REGION Network 2: Block description — Section 3 to 3.2
   // ▄▄▄▄▄▄▄▄▄▄▄▄▄▄▄▄▄▄▄▄▄▄▄▄▄▄▄▄▄▄▄▄▄▄▄▄▄▄▄▄▄▄▄▄
   // 3.     DETAILED BLOCK DESCRIPTION
   // 
   // 
   // This module, FC11001_StdDevValveIsol uses user data types to provide the primary interface to 
   // the module, it also uses direct digital signals to provide an interface for the position feedback 
   // signals and for the fault, safety and interlock signals. It also has a single output signal used to 
   // operate the valve. 
   // 
   // These are the formal module parameters: 
   // 
   //  ――――――――――――――――――――――――――――――――――――――――――
   //  PARAM         FUNCTION                    TYPE      IN-OUT 
   //  ――――――――――――――――――――――――――――――――――――――――――
   //  SYS_SIGNALS      Common system signals              UT21000    In
   //           logic and timing signals for parametric access
   // 
   //  FBK_OPEN     Optional open state positive feedback        Bool      In
   //           (1 = open, 0 = not open) If not required, set 
   //           permanently to _False
   // 
   //  FBK_CLOSED    Optional closed state positive feedback        Bool      In
   //           (1 = closed 0 = not closed) If not required, set 
   //           permanently to _False
   // 
   //  EXT_FAULT     Optional external fault signal for the device     Bool      In
   //           (1 = fault, 0 = healthy). If not required, set 
   //           permanently to _False
   // 
   //  E_STOP        Optional emergency stop (safety) signal        Bool      In
   //           (1 = emergency stop active, 0 = healthy) If not 
   //           required, set permanently to _False
   // 
   //  TRIP        Optional trip signal                  Bool      In
   //           (1 = trip condition active, 0 = healthy) If not 
   //           required, set permanently to _False
   // 
   //  INTERLOCK     Optional interlock signal               Bool      In
   //           (1 = interlock condition active, 0 = healthy) If 
   //           not required, set permanently to _False
   // 
   //  PERMISSIVE      Optional permissive signal             Bool      In
   //           (1 = permissive condition active, 0 = healthy) 
   //           If not required, set permanently to _False
   // 
   //  STATIC_DATA     Data structure that holds the configuration data     UT11001    In
   //           for the device (normally open/closed, limit switch 
   //           and interlock configuration &c.)
   // 
   //  DYNAMIC_DATA      Data structure that holds the live data for the       UT31001    InOut
   //           device (its mode, status and messages and 
   //           any other dynamic information required by the 
   //           module)
   // 
   //  OPERATE        Output to drive the valve to a particular state    Bool      Out
   //           (1 = energised state, 0 = deenergised state)
   //  ――――――――――――――――――――――――――――――――――――――――――
   // 
   // FBK_OPEN, FBK_CLOSED and EXT_FAULT parameters are input signals provided directly from the 
   // device itself (via digital input cards). The OPERATE signal is an output signal (via a digital output 
   // card) that causes the valve to open and close.
   // 
   // The E-STOP parameter is the interface to any safety signal that might apply to the valve; 
   // similarly, the PERMISSIVE, INTERLOCK and TRIP parameters are the links to any such interlock 
   // signals that may be applied to the device.
   // 
   // The STATIC_DATA and DYNAMIC_DATA parameters are UDTs that hold (respectively) the 
   // configuration information and the live data for the device.
   // 
   //  ――――――――――――――――――――――――――――――――――――――――――
   //  PARAM         ASSOCIATED UDT          ASSOCIATED DATA BLOCK
   //  ――――――――――――――――――――――――――――――――――――――――――
   //  STATIC_DATA     UT11001_St_DevValveIsol        DB11001_St_DevValveIsol
   //  DYNAMIC_DATA   UT31001_Dy_DevValveIsol        DB31001_Dy_DevValveIsol
   //  ――――――――――――――――――――――――――――――――――――――――――
   // 
   // 
   // Section 6 contains a full list of all variables within these UDTs.
   // 
   // This arrangement conforms with the PAL philosophy where IO card connections, safety 
   // signals and interlocks have unique formal parameters; all remaining signals are passed as 
   // variables within UDTs, see the Software Design Specification [Ref. 008].
   // 
   // 
   // 
   // ▂▂▂▂▂▂▂▂▂▂▂▂▂▂▂▂▂▂▂▂▂▂▂▂▂▂▂▂▂▂▂▂▂▂▂▂▂▂▂▂▂▂▂▂
   // 3.1      Typical wiring arrangement
   // 
   // 
   // The typical wiring arrangements for a valve with all signals is as follows:
   // 
   //     24VDC  
   //      ─┬─                                ┌───────┐
   //       │                                 │       │  
   //       ├────┬────┐                 │      ─┴─
   //       │       │       │                 │        GND
   //       │       │       │             ┌┻┐ ▁▁
   //    ▁│ ○   ▁│○   ▁│○             │ │▁＼／ NORMALLY 
   //    ▔│ ○   ▔│○   ▔│○             │ │ ／＼   CLOSED
   //     FAULT│ CLOSED│   OPEN│             └┬┘ ▔▔ 
   //       │       │       │                 │     
   //       │       │       │              │  
   //     ┌─┻─┐┌─┻─┐┌─┻─┐          ┌─┻─┐
   //     │  I1.0  ││  I1.1  ││  I1.2  │DI CARD        │  Q1.0 │DO CARD
   //     └─┬─┘└─┬─┘└─┬─┘          └─┬─┘
   //       │       │       │ ┌────────    │
   //       │       │       │ │ FC11001          │
   //       │       │       │ ├──────────┤ │
   //       │       │       │ │          │ │
   //       │       │       │ │           OPERATE ├─┘
   //       │       │       │ │          │
   //       │       │       └─┤ FBK_OPEN        │
   //       │       │         │          │
   //       │       └──────┤ FBK_CLOSED       │
   //       │                 │          │
   //       └───────────┤ EXT_FAULT        │
   //                         │           
   //                         │
   // 
   // 
   // 
   // ▂▂▂▂▂▂▂▂▂▂▂▂▂▂▂▂▂▂▂▂▂▂▂▂▂▂▂▂▂▂▂▂▂▂▂▂▂▂▂▂▂▂▂▂
   // 3.2      Normal operation
   // 
   // 
   // Normal operation can generally be considered the operation of both normally open and normally 
   // closed valves under automatic or manual control (see § 3.5.1 for a full explanation of how 
   // automatic and manual modes are selected). And the mechanisms used to determine the state 
   // of the valve.
   // 
   // 
   // 
   // ▁▁▁▁▁▁▁▁▁▁▁▁▁▁▁▁▁▁▁▁▁▁▁▁▁▁▁▁▁▁▁▁▁▁▁▁▁▁▁▁▁▁▁▁
   // 3.2.1     Opening and closing the valve
   // 
   // 
   // Under automatic mode, the valve is controlled by separate software within the Controller (this 
   // is usually derived from either continuous control logic or sequential control logic and 
   // implemented by the command handling application module).
   // 
   // The result of this software will be to either open the valve or close the valve.
   // 
   // Under manual mode, the valve is controlled directly by the operator via some form of 
   // supervisory system (SCADA or HMI). Again, the result of the manual operator action will be to 
   // either open or close the valve.
   // 
   // There are two signals that, under normal operation, can cause the valve to move to a particular 
   // state, one for automatic mode and one for manual mode, both are passed to the module as 
   // part of the DYNAMIC_DATA parameter (UT31001_Dy_DevValveIsol):
   // 
   // 
   //  DATA STRUCTURE    UT31001_Dy_DevValveIsol
   //  ――――――――――――――――――――――――――――――――――――――――――
   //  SIGNAL         FUNCTION               TYPE     DETAILS
   //  ――――――――――――――――――――――――――――――――――――――――――
   //  ctrl_Aut_OpenClose Causes the valve to open and close     Bool  1 = open the valve
   //            if automatic mode is active            0 = close the valve
   //            (mode_AutMan = 1). If auto mode is 
   //            not active, signal is ignored
   // 
   //  ctrl_Man_OpenClose  Causes the valve to open and close     Bool  1 = open the valve
   //            if manual mode is active             0 = close the valve
   //            (mode_AutMan = 0). If man mode is 
   //            not active, signal is ignored
   //  ――――――――――――――――――――――――――――――――――――――――――
   // 
   // Note:    The above signals specify the required physical state of the valve (either open or 
   //      closed), i.e. it specifies the true state required of the valve irrespective of whether 
   //      the valve is normally open or normally closed. 
   // 
   //      The module will determine whether the OPERATE signal should be activated or 
   //      deactivated to achieve the required state depending on the configuration of the 
   //      valve (either normally open or normally closed).
   // 
   // The operating mode (either automatic or manual) is specified within the DYNAMIC_DATA 
   // parameter UDT (UT31001_Dy_DevValveIsol) mode_AutMan as follows:
   // 
   // 
   //  DATA STRUCTURE    UT31001_Dy_DevValveIsol
   //  ――――――――――――――――――――――――――――――――――――――――――
   //  SIGNAL         FUNCTION               TYPE     DETAILS
   //  ――――――――――――――――――――――――――――――――――――――――――
   //  Mode_AutMan     Identifies the operating mode of     Bool  1 = automatic mode
   //            the valve.                   0 = manual mode
   //  ――――――――――――――――――――――――――――――――――――――――――
   // 
   // It is possible to configure the module such that manual mode is permanently disabled; this uses 
   // the following STATIC_DATA parameter:
   // 
   //  DATA STRUCTURE    UT11001_St_DevValveIsol
   //  ――――――――――――――――――――――――――――――――――――――――――
   //  SIGNAL         FUNCTION               TYPE     DETAILS
   //  ――――――――――――――――――――――――――――――――――――――――――
   //  CONFIG_MAN_DIS     Prevents manual mode being       Bool  1 = no manual mode
   //            activated under all circumstances            0 = manual permitted
   //            device is in auto, Mode_AutMan is 
   //            set permanently to 1
   //  ――――――――――――――――――――――――――――――――――――――――――
   // 
   // If manual mode is disabled (configuration signal CONFIG_MAN_DIS is set to 1), then manual 
   // mode cannot be turned on under any circumstances, the option will be greyed out on the 
   // supervisory system faceplate and the module will constantly set the mode_AutMan signal to 1.
   // 
   // By default the device will be in automatic mode.
   // 
   // The state of the OPERATE parameter is determined by either the ctrl_Aut_OpenClose or 
   // ctrl_Man_OpenClose (depending on whether automatic mode or manual mode is active) and 
   // the type of valve in use (either normally open or normally closed). 
   // 
   // The type of valve is determined by the CONFIG_NO_NC signal specified within the STATIC_DATA 
   // parameter UDT (UT11001_St_DevValveIsol) as follows:
   // 
   // 
   //  DATA STRUCTURE    UT11001_St_DevValveIsol
   //  ――――――――――――――――――――――――――――――――――――――――――
   //  SIGNAL         FUNCTION               TYPE     DETAILS
   //  ――――――――――――――――――――――――――――――――――――――――――
   //  CONFIG_NO_NC      Identifies the type of the valve      Bool  1 = normally open
   //            as either normally open or normally         0 = normally closed
   //            closed.
   // 
   //            A normally closed valve is energised 
   //            to open, deenergised to close.
   // 
   //            A normally open valve is deenergised 
   //            to open and energised to close.
   //  ――――――――――――――――――――――――――――――――――――――――――
   // 
   // The various states of the valve for both automatic/manual and normally open/closed are given 
   // in the following table:
   // 
   // 
   //  ――――――――――――――――――――――――――――――――――――――――――
   //  MODE:   AUTOMATIC MODE (mode_AutMan = 1)
   //  ctrl_Aut_OpenClose ctrl_Man_OpenClose CONFIG_NO_NC   OPERATE  VALVE STATE
   //  ――――――――――――――――――――――――――――――――――――――――――
   //      0         N/A      0 (normally closed)   0      Closed
   //      1         N/A      0 (normally closed)   1      Open
   //      0         N/A      1 (normally open)      1      Closed
   //      1         N/A      1 (normally open)      0      Open
   //  ――――――――――――――――――――――――――――――――――――――――――
   //  MODE:   MANUAL MODE (mode_AutMan = 0)
   //  ctrl_Aut_OpenClose ctrl_Man_OpenClose CONFIG_NO_NC   OPERATE  VALVE STATE
   //  ――――――――――――――――――――――――――――――――――――――――――
   //       N/A          0       0 (normally closed)   0      Closed
   //       N/A          1       0 (normally closed)   1      Open
   //       N/A          0       1 (normally open)      1      Closed
   //       N/A          1       1 (normally open)      0      Open
   //  ――――――――――――――――――――――――――――――――――――――――――
   // 
   // 
   // The module will determine the correct state of the OPERATE parameter based on the operating 
   // mode, required state in that mode and the type of valve in use.
   // 
   // If the valve is in a fault state (see § 3.4), the OPERATE parameter will be set to 0 (deenergised), 
   // irrespective of any other signals.
   // 
   // 
   // 
   // ▁▁▁▁▁▁▁▁▁▁▁▁▁▁▁▁▁▁▁▁▁▁▁▁▁▁▁▁▁▁▁▁▁▁▁▁▁▁▁▁▁▁▁▁
   // 3.2.2     Operation timers
   // 
   // 
   // The module an operation timer used for both opening the valve and for closing the valve.
   // 
   // The timer is loaded with either the opening operation time or closing operation time whenever 
   // the valve is requested to change state. The timer counts down from the loaded value to zero 
   // (the valve can have different times for opening and closing).
   // 
   // The specific operating times are given within the STATIC_DATA parameter 
   // UDT (UT11001_St_DevValveIsol) as follows:
   // 
   // 
   //  DATA STRUCTURE    UT11001_St_DevValveIsol
   //  ――――――――――――――――――――――――――――――――――――――――――
   //  SIGNAL         FUNCTION               TYPE     DETAILS
   //  ――――――――――――――――――――――――――――――――――――――――――
   //  TIME_OPENING_MAX The maximum time required for the     Real     Time in seconds
   //            valve to travel from a closed state to
   //            an open state
   // 
   //  TIME_CLOSING_MAX The maximum time required for the     Real     Time in seconds
   //            valve to travel from an open state to 
   //            a closed state
   //  ――――――――――――――――――――――――――――――――――――――――――
   // 
   // If the timer is running, the elapsed (counting down) time is stored within the DYNAMIC_DATA 
   // parameter UDT (UT31001_Dy_DevValveIsol) as follows:
   // 
   // 
   //  DATA STRUCTURE    UT31001_Dy_DevValveIsol
   //  ――――――――――――――――――――――――――――――――――――――――――
   //  SIGNAL           FUNCTION               TYPE     DETAILS
   //  ――――――――――――――――――――――――――――――――――――――――――
   //  actual_Operating_Timer    The actual elapsed operation time       Real     Time in seconds
   //  ――――――――――――――――――――――――――――――――――――――――――
   // 
   // There is a single operating timer for both opening and closing (opening and closing are mutually 
   // exclusive operations, hence only one timer is needed. The timer is preloaded with either the 
   // opening time preset or the closing time preset prior to the timer starting).
   // 
   // The preset signals TIME_OPENING_MAX and TIME_CLOSING_MAX are the maximum possible 
   // times it can take for the valve to reach the expected position. This should be set to between 
   // 110% and 120% of the normal opening and closing times specified for the valve. For example, 
   // if a valve has a normal opening time of 5 seconds and a normal closing time of 3 seconds, 
   // sensible values for TIME_OPENING_MAX and TIME_CLOSING_MAX would be between 5.5-6.0 s 
   // and 3.3-4.0 s respectively.
   // 
   // A valve will enter a fault state (see § 3.4) if the operation timer counts down to a value of zero 
   // without confirmation that the valve has reached the required state. Such confirmation is 
   // provided by positive feedback from the valve limit switches (or other indicating devices) or 
   // by simulated signal within the module itself (see § 3.2.3).
   // 
   // The operation timer always counts down from a preset value to zero, this is in accordance 
   // with the general requirements and practices of the PAL software.
   // 
   // 
   // 
   // ▁▁▁▁▁▁▁▁▁▁▁▁▁▁▁▁▁▁▁▁▁▁▁▁▁▁▁▁▁▁▁▁▁▁▁▁▁▁▁▁▁▁▁▁
   // 3.2.3     Position feedback signals
   // 
   // 
   // The module can accommodate either none, one or two positive position indication signals:
   // 
   // 
   //    1.  No limit switches         There is no positive indication of the current state 
   //                      of the valve, it is assumed to be in the expected 
   //                      state.
   // 
   //    2.  Closed limit switch only       Positive indication is given for the closed state 
   //                      only. The valve is assumed to be open if the 
   //                      closed signal is inactive.
   // 
   //    3.  Open limit switch only      Positive indication is given for the open state 
   //                      only. The valve is assumed to be closed if the 
   //                      open signal is inactive.
   // 
   //    4.  Open and closed limit switches    Positive indication is given for both states. 
   //                      This allows the true state of the valve to be 
   //                      determined under all circumstances.
   // 
   // There are two configuration signals that determine the position feedback arrangements, these 
   // are stored within the STATIC_DATA parameter UDT as follows:
   // 
   // 
   //  DATA STRUCTURE    UT11001_St_DevValveIsol
   //  ――――――――――――――――――――――――――――――――――――――――――
   //  SIGNAL           FUNCTION              TYPE     DETAILS
   //  ――――――――――――――――――――――――――――――――――――――――――
   //  CONFIG_FBK_OPEN_EN    Indicates that positive feedback for    Bool  1 = open feedback
   //              the open state is present           0 = no feedback
   // 
   //  CONFIG_FBK_CLOSED_EN  Indicates that positive feedback for    Bool  1 = closed feedback
   //              the closed state is present            0 = no feedback
   //  ――――――――――――――――――――――――――――――――――――――――――
   // 
   // If the CONFIG_FBK_OPEN_EN signal is activated (set to 1), the module will use the state of the 
   // signal connected to the FBK_OPEN parameter to determine the open position of the valve. 
   // 
   // If the CONFIG_FBK_OPEN_EN signal is deactivated (set to 0), the module will derive the open 
   // position of the valve such that it matches the requested state of the valve.
   // 
   // Similarly, if the CONFIG_FBK_CLOSED_EN signal is activated (set to 1), the module will use the 
   // state of the signal connected to the FBK_CLOSED parameter to determine the closed position of 
   // the valve. 
   // 
   // If the CONFIG_FBK_CLOSED_EN signal is deactivated (set to 0), the module will derive the 
   // closed position of the valve such that it matches the requested state of the valve.
   // 
   // Where a CONFIG_FBK_OPEN/CLOSED_EN signal is activated (set to 1), a true state on the 
   // associated parameter FBK_OPEN/CLOSED indicates that the valve is in that position, a false 
   // state indicates that the valve is not in that position as follows:
   // 
   //  OPEN SIGNALS  ―――――――――――――――――――――――――――――――――――
   //  CONFIG_FBK_OPEN_EN    FBK_OPEN    MEANING
   //  ――――――――――――――――――――――――――――――――――――――――――
   //       1            0       Not open
   //       1            1       Confirmed open
   //       0          N/A     Internally derived open signal matches
   //                        requested valve state, FBK_OPEN is ignored
   //  ――――――――――――――――――――――――――――――――――――――――――
   //  CLOSED SIGNALS ――――――――――――――――――――――――――――――――――
   //  CONFIG_FBK_CLOSED_EN  FBK_CLOSED  MEANING
   //  ――――――――――――――――――――――――――――――――――――――――――
   //       1            0       Not closed
   //       1            1       Confirmed closed
   //       0          N/A     Internally derived closed signal matches
   //                        requested valve state, FBK_CLOSED is ignored
   //  ――――――――――――――――――――――――――――――――――――――――――   
   // 
   // 
   // 
   // 
   // ▁▁▁▁▁▁▁▁▁▁▁▁▁▁▁▁▁▁▁▁▁▁▁▁▁▁▁▁▁▁▁▁▁▁▁▁▁▁▁▁▁▁▁▁
   // Position status signals
   // 
   // 
   // The true position of the valve is given as status signals:
   // 
   //  DATA STRUCTURE    UT31001_Dy_DevValveIsol
   //  ――――――――――――――――――――――――――――――――――――――――――
   //  SIGNAL          FUNCTION                TYPE     DETAILS
   //  ――――――――――――――――――――――――――――――――――――――――――
   //  status_Closed      Valve is confirmed closed         Bool     1 = closed
   //                                    0 = not closed
   // 
   //  status_Opening      Valve is opening             Bool     1 = opening
   //                                    0 = not opening
   // 
   //  status_Open      Valve is confirmed open         Bool     1 = open
   //                                    0 = not open
   // 
   //  status_Closing     Valve is closing               Bool     1 = closing
   //                                    0 = not closing
   // 
   //  status_Operating      Valve is changing state          Bool     1 = changing state
   //             (either opening or closing)           0 = fixed state
   // 
   //  status_Fault       Valve is in a fault condition          Bool     1 = fault
   //                                    0 = healthy
   //  ――――――――――――――――――――――――――――――――――――――――――   
   // 
   // The standard arrangement is for symbols to show discrete opening and closing symbols; there 
   // are some instances (usually on less sophisticated HMIs) where it is necessary to show only that 
   // the valve is in the process of changing state.
   // 
   // This is achieved through the use of the status_Operating signal (this is active whenever either 
   // status_Opening or status_Closing is active), status_Operating indicates that the valve is either 
   // opening or closing, but does not distinguish which.
   // 
   // 
   // 
   // ▁▁▁▁▁▁▁▁▁▁▁▁▁▁▁▁▁▁▁▁▁▁▁▁▁▁▁▁▁▁▁▁▁▁▁▁▁▁▁▁▁▁▁▁
   // Understanding derived position signals
   // 
   // 
   // Where either the CONFIG_FBK_OPEN_EN or CONFIG_FBK_CLOSED_EN signal is deactivated 
   // (set to 0), the associated position feedback is internally determined by the module according to 
   // the actual state of the valve (determined by the OPERATE parameter and the type of valve in use).
   // 
   // These internally derived signals are themselves configurable and can be set such that the 
   // position feedback signal occurs after a particular percentage of the associated operation timer 
   // has expired.
   // 
   // For the derived FBK_OPEN signal, the configurable percentage signal is TIME_DER_OPEN 
   // stored within the STATIC_DATA parameter. Similarly, for the derived FBK_CLOSED signal, the 
   // configurable percentage signal is TIME_DER_CLOSED, again, stored within the STATIC_DATA 
   // parameter.
   // 
   // The operation of these parameters can be seen below:
   // 
   //     ①                ③
   // │   ┌────────────────┐
   // │   │                │
   // │   │                │      ctrl_Aut_OpenClose
   // │   │                │
   // ┼───┘┈┈┈┈┈┈┈┈┈┈┈┈┈┈┈┈└───────────────
   // 
   // 
   //                      TIME_OPENING_MAX            TIME_CLOSING_MAX
   //      ←         →       ←                →
   // │   ┌──────┐┄┄┐      ┌───────┐┄┄┐
   // │   │      │  ┆      │       │  ┆
   // │   │←    Ａ  →│  ┆      │←      Ｂ    →│  ┆actual_Operating_Timer
   // │   │      │  ┆      │       │  ┆
   // ┼───┘┈┈┈┈┈┈└──┴──────┘┈┈┈┈┈┈┈└──┴────
   //     ╎      ②         ╎       ④
   //     ╎      ╎         ╎       ╎
   //     ↓      ╎         ╎       ↓
   // │───┐      ╎         ╎       ┌───────
   // │   │      ╎         ╎       │
   // │   │      ╎         ╎       │                FBK_CLOSED (derived)
   // │   │      ╎         ╎       │
   // ┼┈┈┈└────────────────────────┘┈┈┈┈┈┈┈
   //     Ｃ      ╎         ╎       Ｆ
   //            ╎         ╎
   //            ╎         ╎
   //            ↓         ↓
   // │          ┌─────────┐
   // │          │         │
   // │          │         │               FBK_OPEN (derived)
   // │          │         │
   // ┼──────────┘┈┈┈┈┈┈┈┈┈└────────────────
   //            Ｄ         Ｅ
   // 
   //   Ａ TIME_DER_OPEN  (95%)
   //   Ｂ TIME_DER_CLOSED  (80%)
   //   Ｃ Closed signal deactivates instantly when the valve is asked to open
   //   Ｄ Open signal activates when actual_Operating_Timer reaches TIME_DER_OPEN 
   //     as a percentage of TIME_OPENING_MAX
   //   Ｅ Open signal deactivates instantly when the valve is asked to close
   //   Ｆ Closed signal activates when actual_Operating_Timer reaches TIME_DER_CLOSED 
   //     as a percentage of TIME_CLOSING_MAX
   // 
   // The figure above assumes a normally closed valve with no position feedback signals (both 
   // CONFIG_FBK_OPEN_EN and CONFIG_FBK_CLOSED_EN are set to 0) operating in automatic mode. 
   // It also assumes that the valve is free to operate without restriction (there are no active interlock 
   // or safety signals).
   // 
   // The valve is initially closed with the derived FBK_CLOSED signal active (1) and the derived 
   // FBK_OPEN signal deactivated (0). At some point 1, the module receives a request to open the 
   // valve.
   // 
   // At this point two things happen, firstly the operation timer starts, with a countdown from the 
   // value TIME_OPENING_MAX, which in this case is 3 seconds. Secondly, the derived FBK_CLOSED 
   // signal is deenergised (indicating the valve is no longer closed).
   // 
   // The simulated opening time (TIME_DER_OPEN) is set to 95%, this means that the derived 
   // FBK_OPEN signal will activate when the actual_Operating_Timer value has counted down for 
   // 95% of the TIME_OPENING_MAX value (i.e. when the timer has counted down to 0.15s or less). 
   // 
   // The exact formula used is:
   // 
   // ┌───────────────────────────────────────────┐
   // │Derived FBK_OPEN=1 when:                                     │
   // │                                 TIME_DER_OPEN        │
   // │actual_Operating_Timer ≤ TIME_OPENING_MAX ─ TIME_OPENING_MAX ╳ --------------------------------        │
   // │                                     100     │
   // └───────────────────────────────────────────┘
   // 
   // This can be seen at point ②, where the derived FBK_OPEN signal activates. The valve now 
   // remains in the open state (FBK_OPEN = 1. FBK_CLOSED = 0) until there is a request to close 
   // the valve, point ③.
   // 
   // Again, at point ③, the module receives a request to close the valve.
   // 
   // At this point two things happen, firstly the operation timer starts, with a countdown from the 
   // value TIME_CLOSING_MAX, which in this case is 4 seconds. Secondly, the derived FBK_OPEN signal 
   // is deenergised (indicating the valve is no longer open).
   // 
   // The simulated closing time (TIME_DER_CLOSED) is set to 80%, this means that the derived 
   // FBK_CLOSED signal will activate when the actual_Operating_Timer value has counted down 
   // for 80% of the TIME_CLOSING_MAX value (i.e. when the timer has counted down to 0.80s or less). 
   // 
   // The exact formula used is:
   // 
   // ┌────────────────────────────────────────────┐
   // │Derived FBK_CLOSED=1 when:                               │
   // │                                 TIME_DER_CLOSED          │
   // │actual_Operating_Timer ≤ TIME_CLOSING_MAX ─ TIME_CLOSING_MAX ╳ ------------------------------------         │
   // │                                     100            │
   // └────────────────────────────────────────────┘
   // 
   // This can be seen at point ④, where the derived FBK_CLOSED signal activates. The valve now 
   // remains in the closed state (FBK_OPEN = 0. FBK_CLOSED = 1) until there is a request a 
   // subsequent request to reopen the valve.
   // 
   // If only one position feedback is derived (the other being an actual signal), then the derived signal 
   // will be generated in exactly the same way as above, the non-derived signal will simply use the 
   // true status of the signal passed as a parameter to the module.
   // 
   // The simulated time signals are passed to the module within the STATIC_DATA parameter 
   // UDT (UT11001_St_DevValveIsol) as follows:
   // 
   //  DATA STRUCTURE    UT11001_St_DevValveIsol
   //  ――――――――――――――――――――――――――――――――――――――――――
   //  SIGNAL        FUNCTION              TYPE     DETAILS
   //  ――――――――――――――――――――――――――――――――――――――――――
   //  TIME_DER_CLOSED           Specifies the percentage of the     Real     Percentage
   //              TIME_OPENING_MAX value that 
   //              must expire before the derived 
   //              FBK_OPEN signal activates.
   // 
   // 
   //  TIME_DER_OPEN             Specifies the percentage of the     Real     Percentage
   //              TIME_CLOSING_MAX value that 
   //              must expire before the derived 
   //              FBK_CLOSED signal activates.
   //  ――――――――――――――――――――――――――――――――――――――――――
   // 
   // Both configuration signals are restricted to the range 0.00-100.00, the default value is 90% for 
   // both open and closed.
   // 
   // 
   // 
   // ▁▁▁▁▁▁▁▁▁▁▁▁▁▁▁▁▁▁▁▁▁▁▁▁▁▁▁▁▁▁▁▁▁▁▁▁▁▁▁▁▁▁▁▁
   // 3.2.4    Recording the last operation time
   // 
   // 
   // The module records the last complete operation time value, it records the actual time taken for 
   // the valve to reach the correct designated position.
   // 
   // For example if the valve received a request to open, and it required 4.8 seconds for the position 
   // feedback to report the correct (open) state, the module would record a value of 4.8 seconds in 
   // the actual_Last_Op_Time value (passed as part of the DYNAMIC_DATA parameter).
   // 
   // Similarly, if the valve were requested to close, and required 6.2 seconds for the position feedback 
   // to report the correct (closed) state, the module would record a value of 6.2 seconds in the 
   // actual_Last_Op_Time value.
   // 
   // The actual_Last_Op_time value forms part of the DYNAMIC_DATA parameter UDT as follows:
   // 
   // 
   //  DATA STRUCTURE    UT31001_Dy_DevValveIsol
   //  ――――――――――――――――――――――――――――――――――――――――――
   //  SIGNAL        FUNCTION              TYPE     DETAILS
   //  ――――――――――――――――――――――――――――――――――――――――――
   //  actual_Last_Op_Time     Stores the actual time taken for     Real     Time in seconds
   //             the valve to achieve the correct 
   //             open or closed state.
   // 
   //             Receives a value of -1.0 if the 
   //             valve did not achieve the correct 
   //             position in the specified 
   //             operation time
   //  ――――――――――――――――――――――――――――――――――――――――――
   // 
   // If the valve does not achieve the requested position (within either the TIME_OPENING_MAX or 
   // TIME_CLOSING_MAX limits), a value of -1.0 is returned as the actual_Last_Op_Time value, 
   // indicating a fault occurred.
   // 
   // 
   // 
   // ▁▁▁▁▁▁▁▁▁▁▁▁▁▁▁▁▁▁▁▁▁▁▁▁▁▁▁▁▁▁▁▁▁▁▁▁▁▁▁▁▁▁▁▁
   // 3.2.5    Detecting position faults
   // 
   // 
   // There are two types of position faults: dynamic and static. 
   // 
   // Dynamic faults occur when the valve is changing state (from open to closed or closed to open) 
   // and fails to achieve the requested position within the relevant operation time.
   // 
   // The dynamic faults are:
   // 
   //    •   Failed to open
   // 
   //    •   Failed to close
   // 
   // Static faults occur when a valve is stable in the requested state (either open or closed) and is 
   // not in the process of moving between states, and some fault occurs such that the position 
   // feedback no longer matches the requested state (e.g. the valve was correctly in the open 
   // state, and then at some point, the open feedback signal was lost without any change being 
   // made to the state of the valve by the module. Such a fault could be a power failure at the valve).
   // 
   // The static faults are:
   // 
   //    •   Failed while open
   // 
   //    •   Failed while closed
   // 
   // If the valve is not equipped with any limit switches (both CONFIG_FBK_OPEN_EN and 
   // CONFIG_FBK_CLOSED_EN are set to 0), then there are no circumstances under which any 
   // position fault can be generated (the valve is always assumed to operate correctly and be in the 
   // required position). 
   // 
   // The following table indicates the conditions under which the various alarms can be generated 
   // for the various position feedback combinations:
   // 
   //  ――――――――――――――――――――――――――――――――――――――――――
   //                    FAILED TO OPEN         FAILED TO CLOSE
   //        LIMIT SWITCH         Opening operation timer    Closing operation timer 
   //      ARRANGEMENT         expired and:                 expired and:
   //  ――――――――――――――――――――――――――――――――――――――――――
   //        No feedback
   //     CONFIG_FBK_OPEN_EN = 0     Not applicable       Not applicable
   //  CONFIG_FBK_CLOSED_EN = 0 
   // 
   //       Open feedback only
   //     CONFIG_FBK_OPEN_EN = 1   Open feedback is INACTIVE     Open feedback is ACTIVE
   //  CONFIG_FBK_CLOSED_EN = 0
   // 
   //      Closed feedback only
   //     CONFIG_FBK_OPEN_EN = 0    Closed feedback is ACTIVE     Closed feedback is INACTIVE
   //  CONFIG_FBK_CLOSED_EN = 1
   // 
   //    Open and closed feedback    Closed feedback is ACTIVE     Closed feedback is INACTIVE
   //     CONFIG_FBK_OPEN_EN = 1          OR                   OR
   //  CONFIG_FBK_CLOSED_EN = 1    Open feedback is INACTIVE     Open feedback is ACTIVE
   //  ――――――――――――――――――――――――――――――――――――――――――
   // 
   //  ――――――――――――――――――――――――――――――――――――――――――
   //                    FAILED WHILE OPEN       FAILED WHILE CLOSED
   //        LIMIT SWITCH         Opening operation timer    Closing operation timer 
   //      ARRANGEMENT         not running and:         not running and:
   //  ――――――――――――――――――――――――――――――――――――――――――
   //        No feedback
   //     CONFIG_FBK_OPEN_EN = 0     Not applicable       Not applicable
   //  CONFIG_FBK_CLOSED_EN = 0 
   // 
   //       Open feedback only
   //     CONFIG_FBK_OPEN_EN = 1   Open feedback is INACTIVE     Open feedback is ACTIVE
   //  CONFIG_FBK_CLOSED_EN = 0
   // 
   //      Closed feedback only
   //     CONFIG_FBK_OPEN_EN = 0    Closed feedback is ACTIVE     Closed feedback is INACTIVE
   //  CONFIG_FBK_CLOSED_EN = 1
   // 
   //    Open and closed feedback    Closed feedback is ACTIVE     Closed feedback is INACTIVE
   //     CONFIG_FBK_OPEN_EN = 1          OR                   OR
   //  CONFIG_FBK_CLOSED_EN = 1    Open feedback is INACTIVE     Open feedback is ACTIVE
   //  ――――――――――――――――――――――――――――――――――――――――――
   // 
   // The OR in the alarm conditions is a logical or, it covers the conditions in which both or neither 
   // limit switches are active; consider the failed to open alarm, if both limits were active, the alarm 
   // would be generated because the closed limit switch is active (irrespective of the state of the 
   // open limit). Similarly, if neither switch were active, the alarm would be generated because the 
   // open limit is inactive (irrespective of the state of the closed limit).
   // 
   // All alarms are reported as message signals, these form part of the DYNAMIC_DATA parameter 
   // UDT as follows:
   // 
   //  DATA STRUCTURE    UT31001_Dy_DevValveIsol
   //  ――――――――――――――――――――――――――――――――――――――――――
   //  SIGNAL          FUNCTION                TYPE     DETAILS
   //  ――――――――――――――――――――――――――――――――――――――――――
   //  msg_FailToOpen     Valve failed to open in the specified     Bool     1 = alarm active
   //             opening operation time                0 = no alarm
   // 
   //  msg_FailToClose     Valve failed to close in the specified     Bool     1 = alarm active
   //             closing operation time               0 = no alarm
   // 
   //  msg_FailWhileOpen  Valve suffered position failure while      Bool     1 = alarm active
   //             in a static OPEN state              0 = no alarm
   // 
   //  msg_FailWhileClosed   Valve suffered position failure while      Bool     1 = alarm active
   //             in a static CLOSED state            0 = no alarm
   //  ――――――――――――――――――――――――――――――――――――――――――
END_REGION

REGION Network 3: Block description — Section 3.3 to 3.5
   // ▂▂▂▂▂▂▂▂▂▂▂▂▂▂▂▂▂▂▂▂▂▂▂▂▂▂▂▂▂▂▂▂▂▂▂▂▂▂▂▂▂▂▂▂
   // 3.3     Fault handling
   // 
   // 
   // There are five fault conditions, four are derived from position faults and one from an external 
   // fault signal:
   // 
   //  ――――――――――――――――――――――――――――――――――――――――――
   //  FAULT         DESCRIPTION                     LATCHING
   //  ――――――――――――――――――――――――――――――――――――――――――
   //  Failed to open      Valve failed to open in the specified               YES
   //             opening operation time
   // 
   //  Failed to close      Valve failed to close in the specified              YES
   //             closing operation time
   // 
   //  Failed while open   Valve suffered position failure while            YES
   //             in a static OPEN state
   // 
   //  Failed while closed   Valve suffered position failure while            YES
   //             in a static CLOSED state
   // 
   //  External fault        The EXT_FAULT signal is active                 NO
   //   ――――――――――――――――――――――――――――――――――――――――――
   // 
   // If any of the above faults are active, the valve will be deenergised (the OPERATE parameter will be 
   // set to 0) and the module will ignore all commands either automatic or manual and will ignore all 
   // interlock conditions.
   // 
   // 
   // ▁▁▁▁▁▁▁▁▁▁▁▁▁▁▁▁▁▁▁▁▁▁▁▁▁▁▁▁▁▁▁▁▁▁▁▁▁▁▁▁▁▁▁▁
   // 3.3.1    Position faults
   // 
   // 
   // All position faults (derived from position feedback signals) are latching fault conditions that  
   // require the operator to issue a reset command, this is usually via a faceplate available at the 
   // supervisory system (SCADA/HMI), but could also be via a hardwired 
   // (pushbutton) signal. 
   // 
   // The reset signal is specified within the DYNAMIC_DATA parameter UDT as follows:        
   // 
   //  DATA STRUCTURE    UT31001_Dy_DevValveIsol
   //  ――――――――――――――――――――――――――――――――――――――――――
   //  SIGNAL         FUNCTION                TYPE     DETAILS
   //  ――――――――――――――――――――――――――――――――――――――――――
   //  mode_Reset        A reset pulse                Bool     1 = reset latched faults
   //            (active for one Controller cycle)            0 = no action
   //  ――――――――――――――――――――――――――――――――――――――――――
   // 
   // 
   // 
   // ▁▁▁▁▁▁▁▁▁▁▁▁▁▁▁▁▁▁▁▁▁▁▁▁▁▁▁▁▁▁▁▁▁▁▁▁▁▁▁▁▁▁▁▁
   // 3.3.2    Resetting position faults
   // 
   // 
   // If a position fault has occurred, and the fault is then reset, the appropriate opening or closing 
   // operation timer will be retriggered, allowing the valve time to achieve the required position.
   // 
   // 
   // 
   // ▁▁▁▁▁▁▁▁▁▁▁▁▁▁▁▁▁▁▁▁▁▁▁▁▁▁▁▁▁▁▁▁▁▁▁▁▁▁▁▁▁▁▁▁
   // 3.3.3    External fault
   // 
   // 
   // The external fault is an optional hardwired signal from the valve, it indicates that the device 
   // itself is registering that there is some problem. Such external fault signals are more commonly 
   // associated with motorised valves (equipped with thermal overload detectors), but may also be 
   // associated with pneumatic or hydraulic operated valves to indicate that the is a 
   // pneumatic/hydraulic system failure.
   // 
   // Such fault signals are generally indicated via a hardwired digital input to the Controller.
   // 
   // The external fault signal (if used) is passed to the module as the parameter: EXT_FAULT .
   // 
   // Any signal connected to the EXT_FAULT parameter must be active high (i.e. the signal must be 
   // set to 1 to indicate the fault condition is present). 
   // 
   // Where a failsafe response signal is used (active when set to 0) is used, it must be inverted at the 
   // EXT_FAULT parameter (similar to the E_STOP signal).
   // 
   // If the EXT_FAULT signal is not required, the input should be set to _False  (again, similar to the
   // E_STOP signal).
   // 
   // The EXT_FAULT signal is non-latching; it does not require a mode_Reset signal to clear the fault. 
   // The external fault will automatically reset whenever the EXT_FAULT signal is set to 0.
   // 
   // 
   // 
   // ▂▂▂▂▂▂▂▂▂▂▂▂▂▂▂▂▂▂▂▂▂▂▂▂▂▂▂▂▂▂▂▂▂▂▂▂▂▂▂▂▂▂▂▂
   // 3.4     Safety and interlocks
   // 
   // 
   // Safety and interlock signals are optional signals, passed as individual parameters to the module 
   // (in the same a manner as IO signals), all such signals are optional, a valve can have all, none or 
   // any combination of the signals.
   // 
   // Safety and interlock signals all act to override the normal operation of the valve (whether in 
   // automatic or manual mode) and force the valve to a particular state.
   // 
   // There is one safety signal and three interlock signals, each having its own formal module 
   // parameter:
   // 
   // 
   //  SAFETY SIGNAL
   //  ――――――――――――――――――――――――――――――――――――――――――
   //  PARAM        FUNCTION                   TYPE     DETAILS 
   //  ――――――――――――――――――――――――――――――――――――――――――
   //  E_STOP       Optional emergency stop (safety) signal       Bool     1 = E-stop active
   //          (1 = emergency stop active, 0 = healthy) If not         0 = healthy
   //          required, set permanently to _False
   //  ――――――――――――――――――――――――――――――――――――――――――
   // 
   // 
   //  INTERLOCK SIGNALS
   //  ――――――――――――――――――――――――――――――――――――――――――
   //  PARAM        FUNCTION                   TYPE     DETAILS  
   //  ――――――――――――――――――――――――――――――――――――――――――
   //  TRIP       Optional trip signal                 Bool     1 = Trip active
   //          (1 = trip condition active, 0 = healthy) If not            0 = healthy
   //          required, set permanently to _False
   // 
   //  INTERLOCK    Optional interlock signal              Bool     1 = Interlock active
   //          (1 = interlock condition active, 0 = healthy) If         0 = healthy
   //          not required, set permanently to _False
   // 
   //  PERMISSIVE     Optional permissive signal            Bool     1 = Permissive active
   //          (1 = permissive condition active, 0 = healthy)           0 = healthy
   //          If not required, set permanently to _False
   //  ――――――――――――――――――――――――――――――――――――――――――
   // 
   // 
   // Each safety and interlock signal has its own configuration signal that must be used to formally 
   // disable the parameter if the signal is not required, these are all within the STATIC_DATA parameter 
   // UDT (UT11001_St_DevValveIsol) as follows:
   // 
   // 
   //  DATA STRUCTURE    UT11001_St_DevValveIsol
   //  ――――――――――――――――――――――――――――――――――――――――――
   //  SIGNAL        FUNCTION              TYPE     DETAILS
   //  ――――――――――――――――――――――――――――――――――――――――――
   //  CONFIG_ESTOP_DIS    Disables the safety signal.        Bool     1 = E_STOP disabled
   //              If set to 1, any signal on the          0 = E_STOP enabled
   //              E_STOP parameter will be 
   //              ignored.
   // 
   //  CONFIG_TRIP_DIS      Disables the trip interlock signal.   Bool     1 = TRIP disabled
   //              If set to 1, any signal on the          0 = TRIP enabled
   //              TRIP parameter will be 
   //              ignored.
   // 
   //  CONFIG_ILOCK_DIS     Disables the interlock signal.    Bool     1 = INTERLOCK disabled
   //              If set to 1, any signal on the          0 = INTERLOCK enabled
   //              INTERLOCK parameter will be 
   //              ignored.
   // 
   //  CONFIG_PERM_DIS   Disables the permissive interlock  Bool     1 = PERMISSIVE disabled
   //              signal. If set to 1, any signal on the       0 = PERMISSIVE enabled
   //              TRIP parameter will be 
   //              ignored.
   //  ――――――――――――――――――――――――――――――――――――――――――
   // 
   // The disable signals are used to formally configure the valve, they allow any supervisory system to 
   // know the correct configuration of the valve and display information accordingly.
   // 
   // 
   // 
   // ▁▁▁▁▁▁▁▁▁▁▁▁▁▁▁▁▁▁▁▁▁▁▁▁▁▁▁▁▁▁▁▁▁▁▁▁▁▁▁▁▁▁▁▁
   // 3.4.1    Safety signal operation
   // 
   // 
   // Safety or emergency stop signals are hardwired signals that remove power from a device forcing 
   // it to a safe state. Such signals act independently of the software (the pressing of an emergency 
   // stop button will physically remove power from the affected devices).
   // 
   // The emergency stop signal is passed to the module as the parameter E_STOP; it informs the 
   // module that the safety signal has been activated and allows the module to adjust the state of 
   // the valve to follow the emergency stop conditions.
   // 
   // When the emergency stop signal is removed, the valve will resume the requested state (with the 
   // appropriate operation timer).
   // 
   // Under emergency stop conditions the valve is always deenergised (both physically by the 
   // hardware and within the software via the actions of this module), the OPERATE output is set to 
   // zero (OPERATE = 0); for a normally closed valve (CONFIG_NO_NC = 0) this means the valve will 
   // close, for a normally open valve (CONFIG_NO_NC = 1), the valve will open.
   // 
   // The emergency stop signal is absolute and will override any other demand made of the valve. 
   // There is no mechanism for bypassing this form of safety signal.
   // 
   // 
   // 
   // ▁▁▁▁▁▁▁▁▁▁▁▁▁▁▁▁▁▁▁▁▁▁▁▁▁▁▁▁▁▁▁▁▁▁▁▁▁▁▁▁▁▁▁▁
   // Typical usage of the E_STOP parameter
   // 
   // 
   // Any safety signal connected to the E_STOP parameter must be active high (i.e. the signal must be 
   // set to 1 to activate the safety signal response). It is often the case, where hardwired emergency 
   // stop signals are used, that the emergency stop condition is activated by the absence of a signal 
   // (a failsafe response) rather than the application of a signal. The module can accommodate this 
   // sense of signal by inverting the E_STOP input:
   // 
   // 
   //                         ┌─────────────
   //      ───────────────────┤ FC11001 
   //                         ├───────────────┤
   //           "ZONEA_ESTOP"              │               │
   //        ────┤╱├──────────┤ E_STOP             │
   //                         │               
   //                         │               
   // 
   // 
   // If no safety signal is used, the parameter is set to the _False tag (note, also that the configuration 
   // signal CONFIG_ESTOP_DIS should also be set to 1):
   // 
   // 
   //                         ┌─────────────
   //      ───────────────────┤ FC11001 
   //                         ├───────────────┤
   //                         │               │
   //                      _False ──┤ E_STOP             │
   //                         │               
   //                         │    
   // 
   // 
   // 
   // ▁▁▁▁▁▁▁▁▁▁▁▁▁▁▁▁▁▁▁▁▁▁▁▁▁▁▁▁▁▁▁▁▁▁▁▁▁▁▁▁▁▁▁▁
   // 3.4.2    Interlock signals
   // 
   // 
   // Interlock signals are a more flexible mechanism for overriding the requested position of the valve. 
   // Interlock signals can be both hardware driven (similar to a safety signal) or can be purely software 
   // derived (unlike a safety signal).
   // 
   // Software derived interlock signals can accommodate more complex and more flexible 
   // arrangements, it would for example, be possible to disable a software derived interlock if the 
   // process were undergoing some particular function, such as cleaning &c.
   // 
   // There are three different types of interlock arrangements:
   // 
   // There are three types of interlock signal:
   // 
   //    1.  INTERLOCK
   //      A simple interlock that is active whenever a set of conditions is true, it will force any 
   //      associated devices to a given safe state.
   // 
   //    2.  PERMISSIVE
   //      Takes no action if a device is in a non-safe state, but once the device is in a safe 
   //      state will prevent a transition to a non-safe state (i.e. will not force a valve to close, 
   //      but once it is closed, will prevent it from re-opening).
   // 
   //    3.  TRIP
   //      A latching interlock, it activates whenever a set of events are true (like an interlock), 
   //      but will not deactivate until the triggering conditions are removed and a reset signal 
   //      has been given (effectively a latching interlock), it will force any associated devices 
   //      to a given safe state.
   // 
   // For any type of interlock, the specified interlock state (or permitted state) can be either open or 
   // closed irrespective of the type of valve (normally open or normally closed); unlike the safety signal, 
   // it does not have to be the deenergised state of the valve.
   // 
   // That said, the most common interlock state is the deenergised state of the valve; i.e. the failsafe 
   // position of the valve.
   // 
   // 
   // 
   // ▁▁▁▁▁▁▁▁▁▁▁▁▁▁▁▁▁▁▁▁▁▁▁▁▁▁▁▁▁▁▁▁▁▁▁▁▁▁▁▁▁▁▁▁
   // Typical usage of interlock signals
   // 
   // 
   // Each type of interlock is passed as its own parameter: TRIP, INTERLOCK or PERMISSIVE. Like the 
   // safety signal (E_STOP), each parameter is active high (i.e. the signal must be set to 1 to activate 
   // the associated interlock signal response). 
   // 
   // Again, it is often the case, where hardwired interlock signals are used, that the condition is 
   // activated by the absence of a signal (i.e. a failsafe response) rather than the application of a 
   // signal. The module can accommodate this sense of signal by inverting the relevant input:
   // 
   // 
   //                         ┌─────────────
   //      ───────────────────┤ FC11001 
   //                         ├───────────────┤
   //        "DB23102_Dy_Perm.V001"     │               │
   //        ────┤╱├──────────┤ PERMISSIVE           │
   //                         │               
   // 
   // If a particular interlock signal is not used, the parameter is set to the _False tag (note also: that 
   // the appropriate configuration signal should also be set to 1: CONFIG_TRIP_DIS, CONFIG_ILOCK_DIS 
   // or CONFIG_PERM_DIS).
   // 
   //                         ┌─────────────
   //      ───────────────────┤ FC11001 
   //                         ├───────────────┤
   //                         │               │
   //                      _False ──┤ TRIP                    │
   //                         │               
   //                         │  
   // 
   // 
   // 
   // ▁▁▁▁▁▁▁▁▁▁▁▁▁▁▁▁▁▁▁▁▁▁▁▁▁▁▁▁▁▁▁▁▁▁▁▁▁▁▁▁▁▁▁▁
   // Configuring the interlock signals
   // 
   // 
   // The state adopted by the valve when a particular interlock is active (TRIP or INTERLOCK) or the 
   // permitted state of the valve (PERMISSIVE) are set individually for each type of interlock signal. 
   // These configuration signals are stored within the STATIC_DATA parameter UDT as follows:
   // 
   // 
   //  DATA STRUCTURE    UT11001_St_DevValveIsol
   // 
   //  ――――――――――――――――――――――――――――――――――――――――――
   //  SIGNAL        FUNCTION              TYPE     DETAILS
   //  ――――――――――――――――――――――――――――――――――――――――――
   //  CONFIG_TRIP_OP_CL   The required state of a valve if     Bool     1 = valve will open
   //              the TRIP signal is active            0 = valve will close
   // 
   //  CONFIG_ILOCK_OP_CL  The required state of a valve if     Bool     1 = valve will open
   //              the INTERLOCK signal is active         0 = valve will close
   // 
   //  CONFIG_PERM_OP_CL  The permitted state of a valve if   Bool     1 = valve may open
   //              the PERMISSIVE signal is active          0 = valve may close
   //  ――――――――――――――――――――――――――――――――――――――――――
   // 
   // For example, if CONFIG_ILOCK_OP_CL is set to 1, the valve will open whenever the INTERLOCK 
   // signal is active (set to 1), this will override any automatic or manual requirement for the valve 
   // (but will not override a safety signal, see below). If CONFIG_ILOCK_OP_CL were set to 0, the 
   // valve would close whenever the INTERLOCK signal was active.
   // 
   // The TRIP signal behaves in exactly the same way as the INTERLOCK signal, but uses 
   // CONFIG_TRIP_OP_CL to set the tripped state of the valve.
   // 
   // Although the TRIP signal requires a reset signal to disengage the interlock conditions, this is 
   // handled by the trip logic itself (usually handled by the trip application modules: FC23200) and 
   // not via this module; simply deactivating the TRIP signal removes the trip state from the valve 
   // and allows it to operate normally.
   // 
   // The PERMISSIVE signal operates in a different way, if CONFIG_PERM_OP_CL were set to 1 
   // (valve is permitted to open), and the valve was currently closed under automatic control when 
   // the PERMISSIVE signal became active, nothing would happen to the valve (it would remain 
   // closed), if the valve then subsequently opened under automatic control, the PERMISSIVE signal
   //  would allow the valve to do so (the valve permitted state is open). However, any attempt by 
   // the automatic system to re-close the valve would not be allowed by the PERMISSIVE signal.
   // 
   // Conversely, if CONFIG_PERM_OP_CL were set to 0 (valve is permitted to close), and the valve 
   // was currently open under automatic control when the PERMISSIVE signal became active, 
   // nothing would happen to the valve (it would remain open), if the valve then subsequently 
   // closed under automatic control, the PERMISSIVE signal would allow the valve to do so (the 
   // valve permitted state is close). However, any attempt by the automatic system to re-open 
   // the valve would not be allowed by the PERMISSIVE signal.
   // 
   // Note:    Where multiple interlock signals are used, it is possible for the different interlocks 
   //      to apply different states to the valve, for example an active TRIP could close 
   //      the valve and an active INTERLOCK open it. Such conflicts are managed by the 
   //      different priorities applied to the interlock signals (see § 3.5).  
   // 
   // 
   // 
   // ▁▁▁▁▁▁▁▁▁▁▁▁▁▁▁▁▁▁▁▁▁▁▁▁▁▁▁▁▁▁▁▁▁▁▁▁▁▁▁▁▁▁▁▁
   // Bypassing interlocks
   // 
   // 
   // Unlike safety signals, all interlock signals can be overridden (or bypassed). The bypass signal is a 
   // single signal that, if active, overrides and deactivates any TRIP, INTERLOCK or PERMISSIVE signal 
   // that may have been activated.
   // 
   // The bypass signal is specified within the DYNAMIC_DATA parameter UDT as follows:
   // 
   // 
   //  DATA STRUCTURE    UT31001_Dy_DevValveIsol
   //  ――――――――――――――――――――――――――――――――――――――――――
   //  SIGNAL         FUNCTION                TYPE     DETAILS
   //  ――――――――――――――――――――――――――――――――――――――――――
   //  mode_BypassOn   Activates bypass mode, if active, any    Bool     1 = bypass mode on
   //            TRIP, INTERLOCK or PERMISSIVE signal          0 = bypass mode off
   //            will be ignored
   //  ――――――――――――――――――――――――――――――――――――――――――
   // 
   // 
   // Bypass mode is a manual operation, generally activated by the operator via a faceplate 
   // available at the supervisory system (SCADA/HMI), or via some hardwired signal, such as 
   // a key-switch.
   // 
   // It is possible to configure the module such that bypass mode is permanently disabled, this uses 
   // the following STATIC_DATA parameter:
   // 
   // 
   //  DATA STRUCTURE    UT11001_St_DevValveIsol
   //  ――――――――――――――――――――――――――――――――――――――――――
   //  SIGNAL       FUNCTION                TYPE     DETAILS
   //  ――――――――――――――――――――――――――――――――――――――――――
   //  CONFIG_BYPASS_DIS    Prevents bypass mode being      Bool     1 = no bypass mode
   //             activated under all circumstances         0 = bypass permitted
   //  ――――――――――――――――――――――――――――――――――――――――――
   //   
   // If bypass mode is disabled (configuration signal CONFIG_BYPASS_DIS is set to 1), then the bypass 
   // mode cannot be turned on under any circumstances, the option will be greyed out on the 
   // supervisory system faceplate and the module will constantly reset the mode_BypassOn signal.
   // 
   // Note:    Safety (E_STOP) signals cannot be bypassed.  
   // 
   //      Similarly, if an interlock signal has a hardwired component (that will override any 
   //      software actions), it also must not be bypassed.
   // 
   // 
   // 
   // ▂▂▂▂▂▂▂▂▂▂▂▂▂▂▂▂▂▂▂▂▂▂▂▂▂▂▂▂▂▂▂▂▂▂▂▂▂▂▂▂▂▂▂▂
   // 3.5     Priority of operation
   // 
   // 
   // The valve is normally controlled by either the automatic system or by manual (operator) control; 
   // however, this operation can be overridden by the various safety and interlock conditions 
   // that can apply to the valve. Each of these operations is assigned a priority and if more than one 
   // is active at the same time, the one with the highest priority will take precedence.
   // 
   // The priorities for the various operations is as follows:
   // 
   // 
   //  ――――――――――――――――――――――――――――――――――――――――――
   //  SIGNAL TYPE       PRIORITY   ASSIGNED VALUE       CAN BE BYPASSED
   //  ――――――――――――――――――――――――――――――――――――――――――
   //  Emergency Stop        High        40                NO
   //  Trip            ↑           30             YES
   //  Interlock            ↑           20             YES
   //  Permissive          ↑           10             YES
   //  Auto/manual control    Low         00                NO
   //  ――――――――――――――――――――――――――――――――――――――――――
   //  High priority signal take precedence over lower priority signals.
   // 
   // Thus, if both the TRIP signal, the INTERLOCK signal and automatic control signal were all active at 
   // the same time, the module will respond only to the TRIP signal (with the higher priority) and will 
   // react accordingly.
END_REGION

REGION Network 4: Block description — Section 3.6 to 4
   // ▂▂▂▂▂▂▂▂▂▂▂▂▂▂▂▂▂▂▂▂▂▂▂▂▂▂▂▂▂▂▂▂▂▂▂▂▂▂▂▂▂▂▂▂
   // 3.6     Operating modes
   // 
   // 
   // This module FC11001_StdDevValveIsol supports various operating modes:
   // 
   //    •   Automatic/manual mode
   // 
   //    •   Interlock bypass mode
   // 
   //    •   Simulation mode
   // 
   //    •   Remote/local mode
   // 
   //    •   Faceplate disabled mode
   // 
   // Examining these in turn:   
   // 
   // 
   // 
   // ▁▁▁▁▁▁▁▁▁▁▁▁▁▁▁▁▁▁▁▁▁▁▁▁▁▁▁▁▁▁▁▁▁▁▁▁▁▁▁▁▁▁▁▁
   // 3.6.1    Automatic and manual modes
   // 
   // 
   // Under normal operation, the valve is in automatic mode and is controlled directly by the 
   // Controller software (usually, sequential or continuous logic); however, it is possible for the 
   // operator to take direct control of the valve by switching it to manual mode.
   // 
   // If manual mode is active, the valve will open and close directly at the command of the operator 
   // and will ignore any automatic mode open and close requests.
   // 
   // If the valve is operating under automatic mode, the manual open/close request follows that of 
   // the automatic mode; this ensures that the valve remains in the same state when initially 
   // switched from automatic mode to manual mode, referred to as bumpless transfer. This approach 
   // minimises any disturbance to the process should the valve be inadvertently switched to manual 
   // mode.
   // 
   // The following data points are associated with automatic/manual mode:
   // 
   //  DATA STRUCTURE    UT11001_St_DevValveIsol
   //  ――――――――――――――――――――――――――――――――――――――――――
   //  SIGNAL         FUNCTION               TYPE     DETAILS
   //  ――――――――――――――――――――――――――――――――――――――――――
   //  CONFIG_MAN_DIS     Prevents manual mode being       Bool  1 = no manual mode
   //            activated under all circumstances            0 = manual permitted
   //  ――――――――――――――――――――――――――――――――――――――――――
   // 
   //  DATA STRUCTURE    UT31001_Dy_DevValveIsol
   //  ――――――――――――――――――――――――――――――――――――――――――
   //  SIGNAL         FUNCTION               TYPE     DETAILS
   //  ――――――――――――――――――――――――――――――――――――――――――
   //  Mode_AutMan     Identifies the operating mode of     Bool  1 = automatic mode
   //            the valve.                   0 = manual mode
   // 
   //  ctrl_Aut_OpenClose Causes the valve to open and close     Bool  1 = open the valve
   //            if automatic mode is active            0 = close the valve
   // 
   //  ctrl_Man_OpenClose  Causes the valve to open and close     Bool  1 = open the valve
   //            if manual mode is active             0 = close the valve
   // 
   //  status_Aut      The valve is in automatic mode      Bool  1 = auto mode
   //                                  0 = no in auto
   // 
   //  status_Man       The valve is in manual mode     Bool  1 = manual mode
   //                                  0 = no in manual
   //  ――――――――――――――――――――――――――――――――――――――――――
   // 
   // Manual mode can only be activated by the operator via a faceplate available at the supervisory 
   // system (SCADA/HMI). 
   // 
   // 
   // 
   // ▁▁▁▁▁▁▁▁▁▁▁▁▁▁▁▁▁▁▁▁▁▁▁▁▁▁▁▁▁▁▁▁▁▁▁▁▁▁▁▁▁▁▁▁
   // 3.6.2    Interlock bypass mode
   // 
   // 
   // All interlock signals (TRIP, INTERLOCK or PERMISSIVE) can be overridden (bypassed). The bypass 
   // signal is a single signal that, if active, overrides and deactivates any TRIP, INTERLOCK or 
   // PERMISSIVE signal that may have been activated.
   // 
   // It is possible to permanently disable the bypass mode for any given valve (preventing the 
   // operator from activating it).
   // 
   // The following data points are associated with the bypass mode:
   // 
   //  DATA STRUCTURE    UT11001_St_DevValveIsol
   //  ――――――――――――――――――――――――――――――――――――――――――
   //  SIGNAL       FUNCTION                TYPE     DETAILS
   //  ――――――――――――――――――――――――――――――――――――――――――
   //  CONFIG_BYPASS_DIS    Prevents bypass mode being      Bool     1 = no bypass mode
   //             activated under all circumstances         0 = bypass permitted
   //  ――――――――――――――――――――――――――――――――――――――――――
   // 
   //  DATA STRUCTURE    UT31001_Dy_DevValveIsol
   //  ――――――――――――――――――――――――――――――――――――――――――
   //  SIGNAL         FUNCTION                TYPE     DETAILS
   //  ――――――――――――――――――――――――――――――――――――――――――
   //  mode_BypassOn   Activates bypass mode, if active, any    Bool     1 = bypass mode on
   //            TRIP, INTERLOCK or PERMISSIVE signal          0 = bypass mode off
   //            will be ignored
   // 
   //  status_BypassOn   Status indication, shows if bypass      Bool     1 = bypass active
   //            mode is active                 0 = bypass inactive
   //  ――――――――――――――――――――――――――――――――――――――――――
   // 
   // Bypass mode can only be activated by the operator usually via a faceplate available at the 
   // supervisory system (SCADA/HMI), alternatively it may be via some form of hardwired signal such 
   // as a key-switch &c. 
   // 
   // If bypass mode is disabled (configuration signal CONFIG_BYPASS_DIS is set to 1), then the bypass 
   // mode cannot be turned on under any circumstances, the option will be greyed out on the 
   // supervisory system faceplate and the module will constantly reset the mode_BypassOn signal.  
   // 
   // 
   // 
   // ▁▁▁▁▁▁▁▁▁▁▁▁▁▁▁▁▁▁▁▁▁▁▁▁▁▁▁▁▁▁▁▁▁▁▁▁▁▁▁▁▁▁▁▁
   // 3.6.3    Simulation mode
   // 
   // 
   // The module can be switched to a simulation mode, in which the position feedback for the valve 
   // is replaced by simulated signals specified by the operator. 
   // 
   // Simulation mode is generally used during testing, but can also be applied in a process 
   // environment if a fault condition is detected; this scenario allows the plant to continue operating 
   // (albeit under some degree of manual control) until the valve is repaired or replaced.
   // 
   // The following data points are associated with the simulation mode:
   // 
   //  DATA STRUCTURE    UT11001_St_DevValveIsol
   //  ――――――――――――――――――――――――――――――――――――――――――
   //  SIGNAL       FUNCTION                TYPE     DETAILS
   //  ――――――――――――――――――――――――――――――――――――――――――
   //  CONFIG_SIM_DIS     Prevents simulation mode being     Bool     1 = no sim mode
   //             activated under all circumstances         0 = sim permitted
   //  ――――――――――――――――――――――――――――――――――――――――――
   // 
   //  DATA STRUCTURE    UT31001_Dy_DevValveIsol
   //  ――――――――――――――――――――――――――――――――――――――――――
   //  SIGNAL         FUNCTION                TYPE     DETAILS
   //  ――――――――――――――――――――――――――――――――――――――――――
   //  mode_SimOn      Activates simulation mode, if active, the   Bool     1 = sim mode on
   //            position feedback will be specified by         0 = sim mode off
   //            mode_SimValue      
   //  mode_SimValue    Specifies the type of simulated position     Int     0 = no feedback
   //            feedback in use                  1 = permanently open
   //                                      2 = permanently closed
   //                                      3 = follow demand
   // 
   //  status_SimOn     Status indication, shows if simulation     Bool     1 = sim active
   //            mode is active                 0 = sim inactive
   //  ――――――――――――――――――――――――――――――――――――――――――
   // 
   // Simulation mode can only be activated by the operator via a faceplate available at the 
   // supervisory system (SCADA/HMI).
   // 
   // If simulation mode is activated, the position feedback for the valve is forced to one of four 
   // states specified by the mode_SimValue variable (this is an enumerated variable):
   // 
   //  ――――――――――――――――――――――――――――――――――――――――――
   //  mode_SimValue  DESCRIPTION               FBK_OPEN FBK_CLOSED
   //  ――――――――――――――――――――――――――――――――――――――――――
   //      0        Permanently disables all position feedback    0     0
   //             (irrespective of any valve position)
   // 
   //      1        Permanently sets valve position to open         1     0
   //             (irrespective of any valve position)
   // 
   //      2        Permanently sets valve position to closed      0     1
   //             (irrespective of any valve position)
   // 
   //      3        Position feedback follows the requested        1/0    0/1
   //             state of the valve              (if valve is open/closed)
   //  ――――――――――――――――――――――――――――――――――――――――――
   // 
   // The mode_SimValue is restricted to the range 0-3.
   // 
   // If simulation mode is disabled (configuration signal CONFIG_SIM_DIS is set to 1), then the 
   // simulation mode cannot be turned on under any circumstances, the option will be greyed out on 
   // the supervisory system faceplate and the module will constantly reset the mode_SimOn signal.
   // 
   // If simulation mode is permitted (CONFIG_SIM_DIS = 0), then setting mode_SimOn to 1 will activate 
   // simulation mode and the any position feedback signals (connected to FBK_OPEN and 
   // FBK_CLOSED) will be overridden according to the value stored in mode_SimValue (see Table above).
   // 
   // The operator can set and adjust the simulation value (mode_SimValue) from the instrument 
   // faceplate on the supervisory system. The simulation value can be adjusted at any time by the 
   // operator (even if simulation mode has not been activated), but will not be applied until 
   // simulation mode is turned on (mode_SimOn = 1). 
   // 
   // If simulation mode is completely disabled (CONFIG_SIM_DIS is set to 1) then the operator will not 
   // be able to adjust the simulated value (mode_SimValue will be greyed out on the faceplate).
   // 
   // 
   // 
   // ▁▁▁▁▁▁▁▁▁▁▁▁▁▁▁▁▁▁▁▁▁▁▁▁▁▁▁▁▁▁▁▁▁▁▁▁▁▁▁▁▁▁▁▁
   // 3.6.4     Remote/local mode
   // 
   // Remote and local operating modes refer to the supervisory system that has control of the 
   // device (i.e. which system can write to the device and change the operating mode of the 
   // device). 
   // 
   // This type of mode is usual present where a plant has a remote central control location (a control 
   // room) that normally controls the device (remote control), but also has a field panel with a local 
   // HMI that an operator in the field can select to take over control of the device (local control) for 
   // maintenance purposes.
   // 
   // The modes are as follows (and are mutually exclusive, only one will be active):
   // 
   //    Remote        Only the remote system in the control room can 
   //                 control the device
   // 
   //    Local            A local system has taken control of the device and the remote 
   //                 system can no longer issue commands to it
   // 
   //    Remote/local disabled   The system does not use remote/local modes and any 
   //      (ALL mode)     supervisory system can issue commands to the device 
   //  
   // Remote/local control is generally handled by the supervisory systems themselves; however, the 
   // supervisory systems need a storage area per device to record which mode that device is in, local 
   // control is often activated by a panel key-switch, that changes the state of several devices from 
   // remote to local (usually all the devices controlled by the local panel).
   // 
   // The module simply identifies the remote/local mode from the mode signals and configuration 
   // signals provided to the module.
   // 
   // For systems that do not use remote/local modes (any supervisory system can control the device, 
   // or control is determined by operator privileges), the remote/local modes can be disabled 
   // (CONFIG_RL_EN is set to zero) and the device is effectively in ALL mode (any system can 
   // control the device).
   // 
   // If remote/local operation is in use, the supervisory system that does not have control will still 
   // display all the information from the device, but will not be able to control the device (it could not 
   // for example, activate simulation mode) and all control function (faceplate functions) will be 
   // greyed out.
   // 
   // The following signals are associated with remote/local/all modes:
   // 
   //  DATA STRUCTURE    UT11001_St_DevValveIsol
   //  ――――――――――――――――――――――――――――――――――――――――――
   //  SIGNAL           FUNCTION            TYPE   DETAILS
   //  ――――――――――――――――――――――――――――――――――――――――――
   //  CONFIG_RL_EN      Allows Remote and Local      Bool    1 = Remote/local selected
   //                 modes to be selected        0 = All mode is active
   // 
   //  DATA STRUCTURE    UT31001_Dy_DevValveIsol
   //  ――――――――――――――――――――――――――――――――――――――――――
   //  SIGNAL           FUNCTION            TYPE   DETAILS
   //  ――――――――――――――――――――――――――――――――――――――――――
   //  mode_RemoteOn       Activates remote mode     Bool    1 = remote mode on, 
   //                 CONFIG_RL_EN must = 1       0 = remote mode off
   // 
   //  mode_LocalOn     Activates local mode          Bool    1 = local mode on, 
   //                 CONFIG_RL_EN must = 1       0 = remote mode off
   // 
   //  status_RemoteOn      Status remote mode on     Bool    1 = remote mode on, 
   //                               0 = remote mode off
   // 
   //  status_LocalOn       Status local mode on      Bool 1 = local mode on, 
   //                               0 = local mode off
   // 
   //  status_RLOff       Status ALL mode is on = 0    Bool 1 = ALL mode on, 
   //                               0 = ALL mode off
   //  ――――――――――――――――――――――――――――――――――――――――――
   //  Block remote/local signals 
   // 
   // By default, remote/local is disabled — ALL mode is selected (CONFIG_RL_EN = 0).
   // 
   // 
   // 
   // 
   // ▁▁▁▁▁▁▁▁▁▁▁▁▁▁▁▁▁▁▁▁▁▁▁▁▁▁▁▁▁▁▁▁▁▁▁▁▁▁▁▁▁▁▁▁
   // 3.6.5     Faceplate disable mode
   // 
   // It is possible to disable the supervisory system faceplate from within the module, the 
   // configuration signal:
   // 
   // 
   //  ――――――――――――――――――――――――――――――――――――――――――
   //  SIGNAL           FUNCTION            TYPE   DETAILS
   //  ――――――――――――――――――――――――――――――――――――――――――
   //  CONFIG_FP_DIS        Disable the supervisory      Bool    1 = Faceplate disabled
   //                 system faceplate           0 = normal
   //  ――――――――――――――――――――――――――――――――――――――――――
   // 
   // If the faceplate is disabled (CONFIG_FP_DIS = 1), the supervisory system must not allow the 
   // device faceplate to be opened (normally achieved by clicking the block icon or device symbol), 
   // this in turn prevents the operator from affecting the device in anyway, it would not, for example, 
   // be possible to put the device into simulation mode.
   // 
   // Similarly, if the faceplate is disabled, the operator will not have access to the mode_Reset signal, 
   // meaning that alternative reset mechanisms must be in place (such as a hardwired pushbutton 
   // for example).
   // 
   //                ━━━   ⬙⬙⬙⬙⬙⬙   ━━━
   // 
   // 
   // 
   // ▄▄▄▄▄▄▄▄▄▄▄▄▄▄▄▄▄▄▄▄▄▄▄▄▄▄▄▄▄▄▄▄▄▄▄▄▄▄▄▄▄▄▄▄
   // 4.     Supervisory system interface
   // 
   // 
   // See the online documentation for this block — select the block in the project tree and press:
   //      SHIFT + F1 or follow the link: https://psop.uk/pal-smds-fc11001-p 
   // 
   // An explanation of the block icons and faceplates available to the supervisory system for this 
   // module is given in section 4 of the SMDS document [Ref. 011].
   // 
   // A downloadable copy of the SMDS (and all other project documentation) is available here:
   // 
   //      https://practicalseries.com/2001-pal/21-project/01-00-docs.html
   // 
   // For this module, the document number is: PS2001-5-2312-fc11001
   // 
   //                ━━━   ⬙⬙⬙⬙⬙⬙   ━━━
END_REGION

REGION Network 5: Block description — Sections 5 to 11
   // ▄▄▄▄▄▄▄▄▄▄▄▄▄▄▄▄▄▄▄▄▄▄▄▄▄▄▄▄▄▄▄▄▄▄▄▄▄▄▄▄▄▄▄▄
   // 5.     PARAMETERS
   // 
   // 
   // The following parameters are associated with the block:
   // 
   //  
   //  ――――――――――――――――――――――――――――――――――――――――――
   //  PARAM         FUNCTION                    TYPE      IN-OUT 
   //  ――――――――――――――――――――――――――――――――――――――――――
   //  SYS_SIGNALS      Common system signals              UT21000    In
   //           logic and timing signals for parametric access
   // 
   //  FBK_OPEN     Optional open state positive feedback        Bool      In
   //           (1 = open, 0 = not open) If not required, set 
   //           permanently to _False
   // 
   //  FBK_CLOSED    Optional closed state positive feedback        Bool      In
   //           (1 = closed 0 = not closed) If not required, set 
   //           permanently to _False
   // 
   //  EXT_FAULT     Optional external fault signal for the device     Bool      In
   //           (1 = fault, 0 = healthy). If not required, set 
   //           permanently to _False
   // 
   //  E_STOP        Optional emergency stop (safety) signal        Bool      In
   //           (1 = emergency stop active, 0 = healthy) If not 
   //           required, set permanently to _False
   // 
   //  TRIP        Optional trip signal                  Bool      In
   //           (1 = trip condition active, 0 = healthy) If not 
   //           required, set permanently to _False
   // 
   //  INTERLOCK     Optional interlock signal               Bool      In
   //           (1 = interlock condition active, 0 = healthy) If 
   //           not required, set permanently to _False
   // 
   //  PERMISSIVE      Optional permissive signal             Bool      In
   //           (1 = permissive condition active, 0 = healthy) 
   //           If not required, set permanently to _False
   // 
   //  STATIC_DATA     Data structure that holds the configuration data     UT11001    In
   //           for the device (normally open/closed, limit switch 
   //           and interlock configuration &c.)
   // 
   //  DYNAMIC_DATA      Data structure that holds the live data for the       UT31001    InOut
   //           device (its mode, status and messages and 
   //           any other dynamic information required by the 
   //           module)
   // 
   //  OPERATE        Output to drive the valve to a particular state    Bool      Out
   //           (1 = energised state, 0 = deenergised state)
   //  ――――――――――――――――――――――――――――――――――――――――――
   // 
   //                ━━━   ⬙⬙⬙⬙⬙⬙   ━━━
   // 
   // 
   // 
   // ▄▄▄▄▄▄▄▄▄▄▄▄▄▄▄▄▄▄▄▄▄▄▄▄▄▄▄▄▄▄▄▄▄▄▄▄▄▄▄▄▄▄▄▄
   // 6.     DATA STRUCTURES AND USAGE
   // 
   // 
   // The block has the following associated data structure:
   // 
   // 
   //  ――――――――――――――――――――――――――――――――――――――――――
   //  DATA STRUCTURE             DESCRIPTION
   //  ――――――――――――――――――――――――――――――――――――――――――
   //  UT01000_St_SysRevision          Revision information for this block    See FC01001
   //  UT01001_St_SysLicence           Licence information for this block  See FC01001
   //  UT21000_Dy_SysSignals           System signals for logic and timing  See FC01001
   // 
   //  UT11001_St_DevValveIsol        Static data that holds the configuration data
   //                     for the device (normally open/closed, limit switch 
   //                     and interlock configuration &c.)
   // 
   //  UT31001_Dy_DevValveIsol          Dynamic data that holds the live data for the
   //                     device (its mode, status and messages and 
   //                     any other dynamic information required by the 
   //                     module)
   // 
   //  ――――――――――――――――――――――――――――――――――――――――――
   // 
   // 
   // 
   // ▂▂▂▂▂▂▂▂▂▂▂▂▂▂▂▂▂▂▂▂▂▂▂▂▂▂▂▂▂▂▂▂▂▂▂▂▂▂▂▂▂▂▂▂
   // 6.1     UT11001_St_DevValveIsol
   // 
   // The static data structure for an isolating valve.
   // 
   // 
   //  UT11001_St_DevValveIsol (full contents)
   //  ――――――――――――――――――――――――――――――――――――――――――
   //  SIGNAL NAME          FUNCTION                     TYPE
   //  ――――――――――――――――――――――――――――――――――――――――――
   //  CONFIG_NO_NC        CONFIG — Normally open or normally closed valve     Bool
   //                      (1 = normally open, 0 = normally closed)
   //  CONFIG_FBK_OPEN_EN    CONFIG — Open feedback is enabled        Bool
   //                      (1 = open feedback, 0 = no feedback)
   //  CONFIG_FBK_CLOSED_EN   CONFIG — Closed feedback is enabled         Bool
   //                      (1 = closed feedback, 0 = no feedback)
   //  CONFIG_ESTOP_DIS     CONFIG — E_STOP signal disabled           Bool
   //                      (1 = E_STOP not used, 0 = in use)
   //  CONFIG_TRIP_DIS      CONFIG — TRIP signal disabled           Bool
   //                      (1 = TRIP not used, 0 = in use)
   //  CONFIG_ILOCK_DIS     CONFIG — INTERLOCK signal disabled        Bool
   //                      (1 = INTERLOCK not used, 0 = in use)
   //  CONFIG_PERM_DIS      CONFIG — PERMISSIVE signal disabled         Bool
   //                      (1 = PERMISSIVE not used, 0 = in use)
   //  CONFIG_TRIP_OP_CL       CONFIG — TRIP state                  Bool
   //                      (1 = open, 0 = close)
   //  CONFIG_ILOCK_OP_CL      CONFIG — INTERLOCK state              Bool
   //                      (1 = open, 0 = close)
   //  CONFIG_PERM_OP_CL       CONFIG — PERMISSIVE permitted state         Bool
   //                      (1 = open, 0 = closed)
   //  CONFIG_FP_DIS               CONFIG — Faceplate is disabled           Bool
   //                      (1 = no Faceplate, 0 = normal)
   //  CONFIG_MAN_DIS              CONFIG — Manual mode is disabled          Bool
   //                      (1 = no manual mode, 0 = normal)
   //  CONFIG_BYPASS_DIS     CONFIG — Bypass mode is disabled           Bool
   //                      (1 = no bypass mode, 0 = normal)
   //  CONFIG_SIM_DIS             CONFIG — Simulation is disabled            Bool
   //                      (1 = no simulation, 0 = normal)
   //  CONFIG_RL_EN       CONFIG — Remote/local mode enabled       Bool
   //                      (1 = enabled, 0 = all mode)
   // 
   //  INFO_TAG          INFORMATION — Instrument ID tag          String[20]
   // 
   //  TIME_OPENING_MAX    TIMER — Initial value of opening operation timer      Real
   //                      (counts down from this value), [seconds]
   //  TIME_CLOSING_MAX       TIMER — Initial value of closing operation timer     Real
   //                      (counts down from this value), [seconds]
   //  TIME_DER_OPEN              TIMER — Percentage of opening timer to expired      Real
   //                      before simulating FBK_OPEN, [percent]
   //  TIME_DER_CLOSED            TIMER — Percentage of closing timer to expired        Real
   //                      before simulating FBK_CLOSED, [percent]
   //  ――――――――――――――――――――――――――――――――――――――――――
   // 
   // 
   // 
   // ▂▂▂▂▂▂▂▂▂▂▂▂▂▂▂▂▂▂▂▂▂▂▂▂▂▂▂▂▂▂▂▂▂▂▂▂▂▂▂▂▂▂▂▂
   // 6.2      UT31001_Dy_DevValveIsol
   // 
   // The static data structure for an isolating valve.
   // 
   // 
   // 
   //  UT31001_Dy_DevValveIsol (full contents)
   //  ――――――――――――――――――――――――――――――――――――――――――
   //  SIGNAL NAME          FUNCTION                     TYPE
   //  ――――――――――――――――――――――――――――――――――――――――――
   //  status_Closed        STATUS — Valve is confirmed closed          Bool
   //                      (1 = closed, 0 = not closed)
   //  status_Open        STATUS — Valve is confirmed open         Bool
   //                      (1 = open, 0 = not open)
   //  status_Closing       STATUS — Valve is closing             Bool
   //                      (1 = closing, 0 = not closing)
   //  status_Opening        STATUS — Valve is opening              Bool
   //                      (1 = opening, 0 = not opening)
   //  status_Operating        STATUS — Valve is changing state           Bool
   //                      (1 = changing state, 0 = fixed state)
   //  status_Fault            STATUS — Valve is in fault              Bool
   //                      (1 = fault present, 0 = healthy)
   //  status_Energised        STATUS — Valve output is on              Bool
   //                      (1 = energised, 0 = deenergised)
   //  status_Aut           STATUS — Automatic mode active           Bool
   //                      (1 = auto mode on, 0 = auto mode off)
   //  status_Man          STATUS — Manual mode active             Bool
   //                      (1 = man mode on, 0 = man mode off)
   //  status_EStop          STATUS — E_STOP safety signal is active         Bool
   //                      (1 = active, 0 = healthy)
   //  status_Trip        STATUS — TRIP signal is active             Bool
   //                      (1 = active, 0 = healthy)
   //  status_Ilock         STATUS — INTERLOCK signal is active            Bool
   //                      (1 = active, 0 = healthy)
   //  status_Perm        STATUS — PERMISSIVE signal is active           Bool
   //                      (1 = active, 0 = healthy)
   //  status_BypassOn        STATUS — Valve is in bypass mode          Bool
   //                      (1 = Simulation mode, 0 = normal)
   //  status_SimOn           STATUS — Valve is in simulation mode               Bool
   //                      (1 = Simulation mode, 0 = normal)
   //  status_RemoteOn       STATUS — Valve is in remote mode                  Bool
   //                      (1 = Remote mode, 0 = normal)
   //  status_LocalOn         STATUS — Valve is in local mode                    Bool
   //                      (1 = Local mode, 0 = normal)
   //  status_RLOff         STATUS — Valve is in ALL mode                   Bool
   //                      (1 = ALL mode, 0 = normal)
   // 
   //  msg_FailToOpen       MESSAGE — Alarm – “Fail to open” is active         Bool
   //  msg_FailToClose       MESSAGE — Alarm – “Fail to close” is active        Bool
   //  msg_FailWhileOpen    MESSAGE — Alarm – “Fail while open” is active      Bool
   //  msg_FailWhileClosed     MESSAGE — Alarm – “Fail while closed” is active   Bool
   //  msg_Flt_External         MESSAGE — Alarm – “external fault" is active      Bool
   // 
   //  mode_AutMan        MODE — Automatic or manual mode selection     Bool
   //                    (1 = auto mode active, 0 = man mode)
   //  mode_BypassOn      MODE — Bypass mode                Bool
   //                    (1 = bypass mode active, 0 = normal)
   //  mode_SimOn         MODE — Simulation mode               Bool
   //                    (1 = sim mode active, 0 = normal)
   //  mode_SimValue       MODE — Simulation value               Int
   //                    (0 = no limits, 1 = always open, 
   //                    2 = always closed, 3 = follow demand)
   //  mode_RemoteOn        MODE — Remote SCADA control enabled       Bool
   //                    (1 = active, 0 = disabled or N/A)
   //  mode_LocalOn         MODE — Local HMI control enabled           Bool
   //                    (1 = active, 0 = disabled or N/A)
   //  mode_Reset        MODE — Fault reset – 1 cycle only           Bool
   //                    (1 = Reset faults, 0 = does nothing)
   //  ctrl_Aut_OpenClose       CONTROL — Auto mode open or close valve     Bool
   //                          (1 = open valve , 0 = close valve)
   //  ctrl_Man_OpenClose      CONTROL — Manual mode open or close valve   Bool
   //                          (1 = open valve , 0 = close valve)
   // 
   //  batch_ID         BATCH — Booking ID (optional for batch operations)   UInt
   // 
   //  actual_Operating_Timer     ACTUAL — Timer value — operating opening/closing  Real
   //                      timer actual value [seconds]
   //  actual_Last_Op_Time       ACTUAL — actual time taken to achieve the last    Real
   //                      good valve position [seconds]
   // 
   //  $derived_fbk_open     INTERNAL — Derived feedback open signal       Bool
   //                          (1 = open , 0 = not open)
   //  $derived_fbk_closed      INTERNAL — Derived feedback closed signal        Bool
   //                          (1 = closed, 0 = not closed)
   //  $sim_fbk_open         INTERNAL — Simulated feedback open signal         Bool
   //                          (1 = open , 0 = not open)
   //  $sim_fbk_closed          INTERNAL — Simulated feedback closed signal      Bool
   //                          (1 = closed, 0 = not closed)
   //  $ctrl_OpenClose       INTERNAL — actual open or close request,         Bool
   //                          incorporates all priorities
   //                         (1 = open valve, 0 = close valve)
   //  $pret_Open             INTERNAL — Edge retention (+ve) rising edge of    Bool
   //                          ctrl_OpenClose (change to opening)
   //  $nret_Close            INTERNAL — Edge retention (-ve) falling edge of        Bool
   //                          ctrl_OpenClose (change to closing)
   //  ――――――――――――――――――――――――――――――――――――――――――
   // 
   // 
   // With the exception of the flowing, all these signals are discussed in the previous sections, the 
   // outstanding items are firstly:
   // 
   //      batch_ID
   // 
   // The batch_ID is not required for normal use; it is only used where a “booking” system is used 
   // (common in batch and routing applications). Such booking applications can acquire the device 
   // if it is free and reserve it for a particular phase of the batch. Batch applications are a topic in 
   // their own right and are discussed separately in the online User Guide.
   // 
   // There are internal working signals (all signals the start with a $ are internal working signals used 
   // by the module). In this instance they are used as follows: 
   //  
   // The $derived_fbk_open and $derived_fbk_closed are the internally derived open and closed 
   // feedback signal used in place of FBK_OPEN and FBK_CLOSED if either CONFIG_FBK_OPEN_EN 
   // or CONFIG_FBK_CLOSED_EN is set to zero.
   // 
   // The $sim_fbk_open and $sim_fbk_closed are the simulated position feedback signal used in 
   // place of FBK_OPEN and FBK_CLOSED if simulation mode is active.
   // 
   // $ctrl_OpenClose is the required state of the valve, it takes into account the auto/manual 
   // requested state and modifies this according to any interlocks, safety signals or faults that 
   // may be present.
   // 
   // The $pret_Open and $nret_Close are edge retention signals used to detect either a rising 
   // (a change to opening) or a falling (a change to closing) edge on the $ctrl_OpenClose signal.
   // 
   // 
   //                ━━━   ⬙⬙⬙⬙⬙⬙   ━━━
   // 
   // 
   // 
   // ▄▄▄▄▄▄▄▄▄▄▄▄▄▄▄▄▄▄▄▄▄▄▄▄▄▄▄▄▄▄▄▄▄▄▄▄▄▄▄▄▄▄▄▄
   // 7.     CONSTANTS AND TEMPORARY (LOCAL) DATA
   // 
   // 
   // 
   // ▂▂▂▂▂▂▂▂▂▂▂▂▂▂▂▂▂▂▂▂▂▂▂▂▂▂▂▂▂▂▂▂▂▂▂▂▂▂▂▂▂▂▂▂
   // 7.1     Constants
   // 
   // 
   // The following constants data is used:
   // 
   //  ――――――――――――――――――――――――――――――――――――――――――
   //  SIGNAL NAME       Value    FUNCTION                  TYPE
   //  ――――――――――――――――――――――――――――――――――――――――――
   //  k_TIME_OP_MIN      0.21      Minimum value for the operation timer     Real
   //  ――――――――――――――――――――――――――――――――――――――――――
   // 
   // 
   // 
   // ▂▂▂▂▂▂▂▂▂▂▂▂▂▂▂▂▂▂▂▂▂▂▂▂▂▂▂▂▂▂▂▂▂▂▂▂▂▂▂▂▂▂▂▂
   // 7.2     Temporary (local) data
   // 
   // 
   // The following temporary data is used:
   // 
   //  ――――――――――――――――――――――――――――――――――――――――――
   //  SIGNAL NAME          FUNCTION                  TYPE
   //  ――――――――――――――――――――――――――――――――――――――――――
   //  revInfo             Revision information for the block         UT01000
   //  licInfo           Licensing information for the block      UT01001
   //  calClosedElapsedTime     Calc - Derived closed signal elapsed time   Real
   //  calOpenElapsedTime       Calc - Derived open signal elapsed time   Real
   //  wrkOpen            Working - open position feedback signal      Bool
   //  wrkClosed         Working - closed position feedback signal   Bool
   //  wrkCtrlPriority40        Working - priority 40 controls the valve      Bool
   //  wrkCtrlPriority30        Working - priority 30 controls the valve      Bool
   //  wrkCtrlPriority20        Working - priority 20 controls the valve      Bool
   //  wrkCtrlPriority10        Working - priority 10 controls the valve      Bool
   //  wrkCtrlPriority00        Working - priority 00 controls the valve      Bool
   //  wrkCtrlAutManOpCl     Working - aut/man open or close request     Bool
   //  wrkTimeFbkOpenSim     Working - Err checked TIME_FBK_OPEN            Real
   //  wrkTimeFbkClosedSim     Working - Err checked TIME_FBK_CLOSED           Real
   //  wrkInt           Working storage area (integer)          Int
   //  wrkReal           Working storage (Real)             Real
   //  wrkDInt           Working storage area (double integer)         DInt
   //  ――――――――――――――――――――――――――――――――――――――――――
   // 
   //                ━━━   ⬙⬙⬙⬙⬙⬙   ━━━
   // 
   // 
   // 
   // ▄▄▄▄▄▄▄▄▄▄▄▄▄▄▄▄▄▄▄▄▄▄▄▄▄▄▄▄▄▄▄▄▄▄▄▄▄▄▄▄▄▄▄▄
   // 8.     BLOCK CALLS AND ASSOCIATIONS
   // 
   // 
   // This section details any blocks which may be called from within this software module (subroutine 
   // functions for example), any partner blocks with which it may be associated (for example a 
   // receive module that is partner with a transmit module &c.). It lists any system functions which 
   // may be called (e.g. reading the real time clock) and any system data types that may be used.
   // 
   // Finally, it lists any special calling requirements for the block (for example, must be called from 
   // within a cyclic interrupt organisation block) and if the block is using “optimised access” (this is 
   // the default arrangement).
   // 
   // 
   // 
   // ▂▂▂▂▂▂▂▂▂▂▂▂▂▂▂▂▂▂▂▂▂▂▂▂▂▂▂▂▂▂▂▂▂▂▂▂▂▂▂▂▂▂▂▂
   // 8.1     Block calls from within this module
   // 
   // 
   // There are no PAL block calls from within this block.
   // 
   // 
   // 
   // ▂▂▂▂▂▂▂▂▂▂▂▂▂▂▂▂▂▂▂▂▂▂▂▂▂▂▂▂▂▂▂▂▂▂▂▂▂▂▂▂▂▂▂▂
   // 8.2     Blocks associated with this module
   // 
   // 
   // This is a stand-alone block and is not associated with any other blocks.
   // 
   // 
   // 
   // ▂▂▂▂▂▂▂▂▂▂▂▂▂▂▂▂▂▂▂▂▂▂▂▂▂▂▂▂▂▂▂▂▂▂▂▂▂▂▂▂▂▂▂▂
   // 8.3     System block calls and system data types
   // 
   // There are no system block calls
   // 
   // 
   // 
   // ▂▂▂▂▂▂▂▂▂▂▂▂▂▂▂▂▂▂▂▂▂▂▂▂▂▂▂▂▂▂▂▂▂▂▂▂▂▂▂▂▂▂▂▂
   // 8.4     Special properties and requirements
   // 
   // 
   // 
   // ▁▁▁▁▁▁▁▁▁▁▁▁▁▁▁▁▁▁▁▁▁▁▁▁▁▁▁▁▁▁▁▁▁▁▁▁▁▁▁▁▁▁▁▁
   // 8.4.1     Block optimisation, IEC compatibility and library conformance
   // 
   // 
   //    •   Block optimisation is ACTIVE for this block.
   // 
   //    •   The block has been checked for IEC compatibility and is compliant.
   // 
   //    •   The block is compatible with all IEC library-conformance module constraints
   // 
   // 
   // 
   // ▁▁▁▁▁▁▁▁▁▁▁▁▁▁▁▁▁▁▁▁▁▁▁▁▁▁▁▁▁▁▁▁▁▁▁▁▁▁▁▁▁▁▁▁
   // 8.4.2     Calling requirements
   // 
   // 
   // There are no special calling requirements for this block.
   // 
   //                ━━━   ⬙⬙⬙⬙⬙⬙   ━━━
   // 
   // 
   // 
   // ▄▄▄▄▄▄▄▄▄▄▄▄▄▄▄▄▄▄▄▄▄▄▄▄▄▄▄▄▄▄▄▄▄▄▄▄▄▄▄▄▄▄▄▄
   // 9.     EXAMPLE USAGE
   // 
   // 
   // The following shows a typical deployment of FC11001:
   // 
   //                         ┌─────────────
   //      ───────────────────┤ FC11001 
   //                         ├───────────────┤
   //    "DB21001_DY_StdGlobalData".SysSignals ─┤ SYS_SIGNALS            %Q1.0
   //                         │             OPERATE ├─  "V001_OPR"
   //                   %I1.2     │               │
   //                 "V001_FBK_OPEN" ─┤ FBK_OPEN             │
   //                         │               │
   //                   %I1.1     │               │
   //               "V001_FBK_CLOSED" ─┤ FBK_CLOSED            │
   //                         │               │
   //            %I1.0            │               │
   //           "V001_FAULT"             │               │
   //        ────┤╱├──────────┤ EXT_FAULT                │
   //                         │               │
   //            %I1.4            │               │
   //          "ZONEA_ESTOP"               │               │
   //        ────┤╱├──────────┤ E_STOP                │
   //                         │               │
   //                    "_False" ─┤ TRIP                    │
   //                         │               │
   //            "DB23002_Dy_ILock.V001"─┤ INTERLOCK             │
   //                         │               │
   //                    "_False" ─┤ PERMISSIVE            │
   //                         │               │
   //                         │               │
   //                         │               │
   //         "DB11001_St_DevValveIsol".V001 ─┤ STATIC_DATA             │
   //                         │
   //         "DB31001_Dy_DevValveIsol".V001 ─┤ DYNAMIC_DATA
   //                         │
   //                         │
   //                                         │
   //                                ─────────┘
   // 
   // 
   //               ━━━   ⬙⬙⬙⬙⬙⬙   ━━━
   // 
   // 
   // 
   // ▄▄▄▄▄▄▄▄▄▄▄▄▄▄▄▄▄▄▄▄▄▄▄▄▄▄▄▄▄▄▄▄▄▄▄▄▄▄▄▄▄▄▄▄
   // 10.     TEST AND VERIFICATION PATH
   // 
   // 
   // The following diagram shows the full test and verification path for the formal release of each 
   // version of the software module. See the Test Plan [Ref. 003] for full details, available here:
   //         https://psop.uk/pal-tp-p
   // 
   // 
   //         FC11001-T001         FC11001-T002
   // 
   //     Test version: 000.801     Test version: 001.801
   //  Released version: 001.000     Released version: 002.000
   // Released commit: D0009    Released commit: D0011
   // 
   //        SCR      SMT              SCV     
   // ＿＿＿＿＿＿┌┐＿＿ ▛▜ ＿＿＿＿＿＿＿＿＿＿＿＿╓╖＿＿
   //       └┘   ▙▟             ╙╜  
   // Initial test           Comments standardised
   // 
   // Initial test to release the      Comments updated & 
   // module following the      minor typographical 
   // development stage.       corrections
   // Full SMT              SCV only
   // 
   // 
   // Where:
   // ――――――――――――――――――――――――――――――――――――――――――――
   //  SCR    Source Code Review      A visual inspection of the software to ensure it has been written  
   // ┌┐             to the correct standards, uses the correct structures within the
   // └┘             software and is generally suitable for deployment.               
   // 
   //  SMT Software Module Test    A full and detailed test of an individual software module in
   //   ▛▜              isolation; such testing requires that all branches of the 
   //   ▙▟              software are tested. 
   // 
   //                It tests all the interfaces to the module, any data recorded or 
   //                stored by the module, all error and exception handling functions 
   //                and tests all timed and interrupt driven operations.
   // 
   //  SCV Software Compatibility     A mechanism for verifying that no executable code software 
   // ╓╖    Verification          changes have been made to a module following changes to
   // ╙╜             comment fields.
   // 
   //                Allows typographical errors &c. to be corrected without forcing 
   //                a full SMT on a module that has not functionally changed.
   // ――――――――――――――――――――――――――――――――――――――――――――
   // 
   // An SCV can only be performed on a module that has at some point previously, successfully 
   // completed both an SCR and SMT. Where an SCV is implemented, it replaces the requirement for 
   // both the SCR and the SMT for the test iteration in question.
   // 
   //                ━━━   ⬙⬙⬙⬙⬙⬙   ━━━
   // 
   // 
   // ██████████████ █ █ █ █  END   █ █ █ █ ██████████████
END_REGION

